PROGRAM MAIN
VAR
	nCounter : INT;
END_VAR

nCounter := nCounter +1;

END_PROGRAM

(* stored: Version 1.1.0.1, ProductVersion 3.1.4024.12
   POU MAIN: Id {4b0696f6-af6c-46f9-8f33-29d4909b2e53}, SpecialFunc None *)
